# EPICS substitutions: apps/pcMonitorApp/src/pcMonitor.subs
file pcMonitor.template {

{ BOOTPC     	= "PC-MONITOR"
 }

}
